Universal Robots PolyScope program: tool_change_JF.urp

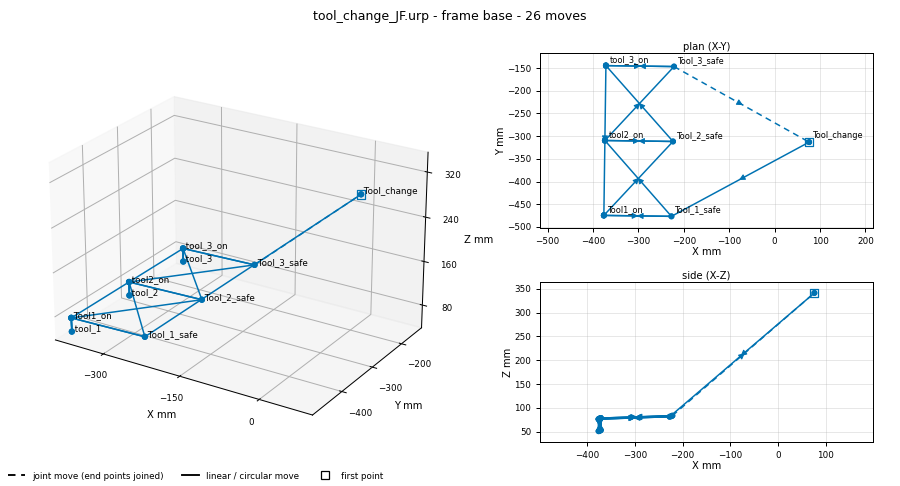
[picture p0: tool path of tool_change_JF.urp in frame base, 26 of 26 moves have a stored position in this frame; points joined in program order, loops and branches not executed]
Program tool_change_JF (installation=default directory=/programs/usbdisk/Ur-Program/Tool-change createdIn=3.10.1.76190 lastSavedIn=3.10.1.76190 robotSerialNumber=2018359886)
Calibrated DH parameters: a=[-0.000111, -0.180064, -0.391564, 0.000025, 0.000035, 0]; d=[0.089308, 162.079685, -160.155007, -1.814221, 0.094754, 0.082578]; alpha=[1.569707, -0.002379, 0.010338, 1.570474, -1.569894, 0]; deltaTheta=[0.000021, -1.133914, 1.184629, -0.050828, 0.000017, 0.000075]
Robot Program (runOnlyOnce=false)
  MoveJ speed 60 deg/s, acceleration 80 deg/s^2 (useActiveTCP=false) tcp=TCP_Schunk
    Waypoint Tool_change: TCP in base x=75.984 y=-313.148 z=341.083 mm, rx=0 ry=0.0001 rz=-0.2764 rad; joints [-56.431, -64.397, -114.786, -90.868, 90.559, 49.445] deg; flange x=75.993 y=-313.149 z=397.063 mm, rx=-0.4326 ry=-3.1115 rz=0 rad
  Set NoAction tcp=TCP_Schunk
  If Old_Tool≟1
    If Tool1≟ False
      MoveL speed 250 mm/s, acceleration 1200 mm/s^2 (useActiveTCP=false) tcp=TCP_Schunk; feature=Base
        Waypoint Tool_1_safe: TCP in base x=-227.333 y=-476.653 z=81.63 mm, rx=0.0068 ry=0.0007 rz=-0.2531 rad; joints [-103.501, -109.067, -114.718, -46.64, 90.288, 1.376] deg; flange x=-227.336 y=-477.036 z=137.608 mm, rx=-0.3963 ry=-3.1157 rz=-0.0106 rad
        Waypoint Tool1_on: TCP in base x=-376.178 y=-474.572 z=76.626 mm, rx=0.0067 ry=0.0008 rz=-0.2532 rad; joints [-117.914, -117.909, -101.757, -50.724, 90.219, -13.088] deg; flange x=-376.178 y=-474.953 z=132.605 mm, rx=-0.3964 ry=-3.1156 rz=-0.0106 rad
        Waypoint tool_1: TCP in base x=-376.117 y=-474.426 z=51.327 mm, rx=0.0068 ry=0.0008 rz=-0.2813 rad; joints [-117.918, -120.188, -102.793, -47.413, 90.203, -11.459] deg; flange x=-376.123 y=-474.809 z=107.305 mm, rx=-0.4402 ry=-3.1097 rz=-0.0106 rad
      Set DigitalOutput pin=digital_out[6]; digitalValue=0
      Set DigitalOutput (payload=0.78 tcpAsCog=false) tcp=TCP_Schunk; pin=digital_out[7]; digitalValue=1
      Wait Sleep waitTime=0.5
      Set DigitalOutput pin=digital_out[7]; digitalValue=0
      MoveL speed 250 mm/s, acceleration 1200 mm/s^2 (useActiveTCP=false) tcp=TCP_Schunk; feature=Base
        Waypoint Tool1_on: TCP in base x=-376.178 y=-474.572 z=76.626 mm, rx=0.0067 ry=0.0008 rz=-0.2532 rad; joints [-117.914, -117.909, -101.757, -50.724, 90.219, -13.088] deg; flange x=-376.178 y=-474.953 z=132.605 mm, rx=-0.3964 ry=-3.1156 rz=-0.0106 rad
    Else 
      Popup Message (haltProgram=false message=something blocking tool 1 storage inputType=Text)
  'skipping tool 0-> No tool on robot'
  If Old_Tool≟2
    If Tool2≟ False
      MoveL speed 250 mm/s, acceleration 1200 mm/s^2 (useActiveTCP=false) tcp=TCP_Schunk; feature=Base
        Waypoint Tool_2_safe: TCP in base x=-223.878 y=-311.698 z=82.74 mm, rx=0.0071 ry=0.0008 rz=-0.2532 rad; joints [-109.097, -91.747, -136.674, -42.016, 90.222, -4.143] deg; flange x=-223.881 y=-312.102 z=138.719 mm, rx=-0.3964 ry=-3.1156 rz=-0.0112 rad
        Waypoint tool2_on: TCP in base x=-373.864 y=-309.584 z=77.743 mm, rx=0.0071 ry=0.0007 rz=-0.2531 rad; joints [-127.272, -104.754, -121.779, -43.843, 90.117, -22.366] deg; flange x=-373.871 y=-309.984 z=133.721 mm, rx=-0.3963 ry=-3.1157 rz=-0.0111 rad
        Waypoint tool_2: TCP in base x=-373.87 y=-309.418 z=52.275 mm, rx=0.0069 ry=0.0008 rz=-0.2766 rad; joints [-127.289, -107.78, -122.985, -39.603, 90.088, -21.011] deg; flange x=-373.875 y=-309.809 z=108.254 mm, rx=-0.4329 ry=-3.1107 rz=-0.0109 rad
      Set DigitalOutput pin=digital_out[6]; digitalValue=0
      Set DigitalOutput (payload=0.78 tcpAsCog=false) tcp=TCP_Schunk; pin=digital_out[7]; digitalValue=1
      Wait Sleep waitTime=0.5
      Set DigitalOutput pin=digital_out[7]; digitalValue=0
      MoveL speed 250 mm/s, acceleration 1200 mm/s^2 (useActiveTCP=false) tcp=TCP_Schunk; feature=Base
        Waypoint tool2_on: TCP in base x=-373.864 y=-309.584 z=77.743 mm, rx=0.0071 ry=0.0007 rz=-0.2531 rad; joints [-127.272, -104.754, -121.779, -43.843, 90.117, -22.366] deg; flange x=-373.871 y=-309.984 z=133.721 mm, rx=-0.3963 ry=-3.1157 rz=-0.0111 rad
    Else 
      Popup Message (haltProgram=false message=something blocking tool 2 inputType=Text)
  If Old_Tool≟3
    If Tool3≟ False
      MoveL speed 250 mm/s, acceleration 1200 mm/s^2 (useActiveTCP=false) tcp=TCP_Schunk; feature=Base
        Waypoint Tool_3_safe: TCP in base x=-221.626 y=-146.719 z=83.867 mm, rx=0.0071 ry=0.0008 rz=-0.2532 rad; joints [-122.112, -71.21, -152.288, -46.895, 90.2, -17.154] deg; flange x=-221.627 y=-147.119 z=139.846 mm, rx=-0.3964 ry=-3.1156 rz=-0.0111 rad
        Waypoint tool_3_on: TCP in base x=-371.646 y=-144.64 z=78.859 mm, rx=0.0071 ry=0.0007 rz=-0.2532 rad; joints [-142.715, -94.273, -134.837, -41.189, 90.022, -37.761] deg; flange x=-371.65 y=-145.041 z=134.838 mm, rx=-0.3964 ry=-3.1156 rz=-0.0112 rad
        Waypoint tool_3: TCP in base x=-371.626 y=-144.442 z=53.376 mm, rx=0.0071 ry=0.0007 rz=-0.2532 rad; joints [-142.741, -98.093, -136.292, -35.914, 89.98, -37.755] deg; flange x=-371.631 y=-144.842 z=109.354 mm, rx=-0.3965 ry=-3.1156 rz=-0.0111 rad
      Set DigitalOutput pin=digital_out[6]; digitalValue=0
      Set DigitalOutput (payload=0.78 tcpAsCog=false) tcp=TCP_Schunk; pin=digital_out[7]; digitalValue=1
      Wait Sleep waitTime=0.5
      Set DigitalOutput pin=digital_out[7]; digitalValue=0
      MoveL speed 250 mm/s, acceleration 1200 mm/s^2 (useActiveTCP=true) feature=Base
        Waypoint tool_3_on: TCP in base x=-371.646 y=-144.64 z=78.859 mm, rx=0.0071 ry=0.0007 rz=-0.2532 rad; joints [-142.715, -94.273, -134.837, -41.189, 90.022, -37.761] deg; flange x=-371.65 y=-145.041 z=134.838 mm, rx=-0.3964 ry=-3.1156 rz=-0.0112 rad
    Else 
      Popup Message (haltProgram=false message=something blocking tool3 storage inputType=Text)
  If New_Tool≟1
    If Tool1≟ True
      MoveL speed 250 mm/s, acceleration 1200 mm/s^2 (useActiveTCP=false) tcp=TCP_Schunk; feature=Base
        Waypoint Tool1_on: TCP in base x=-376.178 y=-474.572 z=76.626 mm, rx=0.0067 ry=0.0008 rz=-0.2532 rad; joints [-117.914, -117.909, -101.757, -50.724, 90.219, -13.088] deg; flange x=-376.178 y=-474.953 z=132.605 mm, rx=-0.3964 ry=-3.1156 rz=-0.0106 rad
        Waypoint tool_1: TCP in base x=-376.117 y=-474.426 z=51.327 mm, rx=0.0068 ry=0.0008 rz=-0.2813 rad; joints [-117.918, -120.188, -102.793, -47.413, 90.203, -11.459] deg; flange x=-376.123 y=-474.809 z=107.305 mm, rx=-0.4402 ry=-3.1097 rz=-0.0106 rad
      Set DigitalOutput (payload=1.41 tcpAsCog=false) tcp=TCP_Tool1; pin=digital_out[6]; digitalValue=1
      Wait Sleep waitTime=0.5
      MoveL speed 250 mm/s, acceleration 1200 mm/s^2 (useActiveTCP=false) tcp=TCP_Schunk; feature=Base
        Waypoint Tool1_on: TCP in base x=-376.178 y=-474.572 z=76.626 mm, rx=0.0067 ry=0.0008 rz=-0.2532 rad; joints [-117.914, -117.909, -101.757, -50.724, 90.219, -13.088] deg; flange x=-376.178 y=-474.953 z=132.605 mm, rx=-0.3964 ry=-3.1156 rz=-0.0106 rad
        Waypoint Tool_1_safe: TCP in base x=-227.333 y=-476.653 z=81.63 mm, rx=0.0068 ry=0.0007 rz=-0.2531 rad; joints [-103.501, -109.067, -114.718, -46.64, 90.288, 1.376] deg; flange x=-227.336 y=-477.036 z=137.608 mm, rx=-0.3963 ry=-3.1157 rz=-0.0106 rad
    Else 
      Popup Message (haltProgram=false message=tool 1 not in place inputType=Text)
  If New_Tool≟2
    If Tool2≟ True
      MoveL speed 250 mm/s, acceleration 1200 mm/s^2 (useActiveTCP=false) tcp=TCP_Schunk; feature=Base
        Waypoint tool2_on: TCP in base x=-373.864 y=-309.584 z=77.743 mm, rx=0.0071 ry=0.0007 rz=-0.2531 rad; joints [-127.272, -104.754, -121.779, -43.843, 90.117, -22.366] deg; flange x=-373.871 y=-309.984 z=133.721 mm, rx=-0.3963 ry=-3.1157 rz=-0.0111 rad
        Waypoint tool_2: TCP in base x=-373.87 y=-309.418 z=52.275 mm, rx=0.0069 ry=0.0008 rz=-0.2766 rad; joints [-127.289, -107.78, -122.985, -39.603, 90.088, -21.011] deg; flange x=-373.875 y=-309.809 z=108.254 mm, rx=-0.4329 ry=-3.1107 rz=-0.0109 rad
      Set DigitalOutput (payload=1.87 tcpAsCog=false) tcp=TCP_Tool2; pin=digital_out[6]; digitalValue=1
      Set SingleDigitalPulseActionState SingleDigitalPulseActionState(hiPulseInSeconds=0.5, pin=digital_out[0])
      Wait Sleep waitTime=0.5
      MoveL speed 250 mm/s, acceleration 1200 mm/s^2 (useActiveTCP=false) tcp=TCP_Schunk; feature=Base
        Waypoint tool2_on: TCP in base x=-373.864 y=-309.584 z=77.743 mm, rx=0.0071 ry=0.0007 rz=-0.2531 rad; joints [-127.272, -104.754, -121.779, -43.843, 90.117, -22.366] deg; flange x=-373.871 y=-309.984 z=133.721 mm, rx=-0.3963 ry=-3.1157 rz=-0.0111 rad
        Waypoint Tool_2_safe: TCP in base x=-223.878 y=-311.698 z=82.74 mm, rx=0.0071 ry=0.0008 rz=-0.2532 rad; joints [-109.097, -91.747, -136.674, -42.016, 90.222, -4.143] deg; flange x=-223.881 y=-312.102 z=138.719 mm, rx=-0.3964 ry=-3.1156 rz=-0.0112 rad
    Else 
      Popup Message (haltProgram=false message=tool 2 not in place inputType=Text)
  If New_Tool≟3
    If Tool3≟ True
      MoveL speed 250 mm/s, acceleration 1200 mm/s^2 (useActiveTCP=false) tcp=TCP_Schunk; feature=Base
        Waypoint tool_3_on: TCP in base x=-371.646 y=-144.64 z=78.859 mm, rx=0.0071 ry=0.0007 rz=-0.2532 rad; joints [-142.715, -94.273, -134.837, -41.189, 90.022, -37.761] deg; flange x=-371.65 y=-145.041 z=134.838 mm, rx=-0.3964 ry=-3.1156 rz=-0.0112 rad
        Waypoint tool_3: TCP in base x=-371.626 y=-144.442 z=53.376 mm, rx=0.0071 ry=0.0007 rz=-0.2532 rad; joints [-142.741, -98.093, -136.292, -35.914, 89.98, -37.755] deg; flange x=-371.631 y=-144.842 z=109.354 mm, rx=-0.3965 ry=-3.1156 rz=-0.0111 rad
      Set DigitalOutput (payload=1.28 tcpAsCog=false) tcp=TCP_Tool3; pin=digital_out[6]; digitalValue=1
      Wait Sleep waitTime=0.5
      MoveL speed 250 mm/s, acceleration 1200 mm/s^2 (useActiveTCP=false) tcp=TCP_Schunk; feature=Base
        Waypoint tool_3_on: TCP in base x=-371.646 y=-144.64 z=78.859 mm, rx=0.0071 ry=0.0007 rz=-0.2532 rad; joints [-142.715, -94.273, -134.837, -41.189, 90.022, -37.761] deg; flange x=-371.65 y=-145.041 z=134.838 mm, rx=-0.3964 ry=-3.1156 rz=-0.0112 rad
        Waypoint Tool_3_safe: TCP in base x=-221.626 y=-146.719 z=83.867 mm, rx=0.0071 ry=0.0008 rz=-0.2532 rad; joints [-122.112, -71.21, -152.288, -46.895, 90.2, -17.154] deg; flange x=-221.627 y=-147.119 z=139.846 mm, rx=-0.3964 ry=-3.1156 rz=-0.0111 rad
    Else 
      Popup Message (haltProgram=false message=tool  3 not in place inputType=Text)
  MoveJ speed 60 deg/s, acceleration 80 deg/s^2 (useActiveTCP=true)
    Waypoint Tool_change: TCP in base x=75.984 y=-313.148 z=341.083 mm, rx=0 ry=0.0001 rz=-0.2764 rad; joints [-56.431, -64.397, -114.786, -90.868, 90.559, 49.445] deg; flange x=75.993 y=-313.149 z=397.063 mm, rx=-0.4326 ry=-3.1115 rz=0 rad
  Old_Tool := New_Tool
